// TIA Portal V20 export
TYPE "type_emRelations_em11_sequence"
// stored: Access Published, Namespace Unit1
   STRUCT
      weightCheck : Struct
         jobs : "LAF_typeJobs";
         sequence : "LAF_typeSequence";
         selectJobStatus { S7_SetPoint := 'True'} : Array[0..10] of "LAF_typeJobStatus";
         "step" : "LER_typeStep";
         jobInterface : Struct
            loadJob2 : "LER_typeJobInterface";
            inspectionJob3 : "LER_typeJobInterface";
            unloadJob4 : "LER_typeJobInterface";
         END_STRUCT;
         homeCheck : Struct
            partNoDetect { ExternalWritable := 'False'} : Bool;
            partDetect { ExternalWritable := 'False'} : Bool;
         END_STRUCT;
      END_STRUCT;
   END_STRUCT;
   // // weightCheck."step".action1[101] : Step[101] : JOB[1] Condition
   // // weightCheck."step".action1[110] : Step[110] : Stage Lift Down
   // // weightCheck."step".action1[190] : Step[190] : JOB[1] Step End
   // // weightCheck."step".action1[201] : Step[201] : JOB[2] Condition
   // // weightCheck."step".action1[210] : Step[210] : Weight Check Loading Request => Transfer PP Right
   // // weightCheck."step".action1[230] : Step[230] : Stage Lift Up
   // // weightCheck."step".action1[240] : Step[240] : Weight Check Loading Check => Transfer PP Right
   // // weightCheck."step".action1[250] : Step[250] : Weight Check JR Detection Check
   // // weightCheck."step".action1[290] : Step[290] : JOB[2] Step End
   // // weightCheck."step".action1[301] : Step[301] : JOB[3] Condition
   // // weightCheck."step".action1[310] : Step[310] : Stage Lift Down
   // // weightCheck."step".action1[330] : Step[330] : Weight Check
   // // weightCheck."step".action1[390] : Step[390] : JOB[3] Step End
   // // weightCheck."step".action1[401] : Step[401] : JOB[4] Condition
   // // weightCheck."step".action1[410] : Step[410] : Stage Lift Up
   // // weightCheck."step".action1[430] : Step[430] : Weight Check Unloading Request => JR Unload P&P
   // // weightCheck."step".action1[431] : Step[431] : Weight Check Unloading Check => JR Unload P&P
   // // weightCheck."step".action1[480] : Step[480] : Stage Lift Down
   // // weightCheck."step".action1[490] : Step[490] : JOB[4] Step End
   // // weightCheck."step".transition1[101] : Step[101] : JOB[1] Condition
   // // weightCheck."step".transition1[110] : Step[110] : Stage Lift Down
   // // weightCheck."step".transition1[190] : Step[190] : JOB[1] Step End
   // // weightCheck."step".transition1[201] : Step[201] : JOB[2] Condition
   // // weightCheck."step".transition1[210] : Step[210] : Weight Check Loading Request => Transfer PP Right
   // // weightCheck."step".transition1[230] : Step[230] : Stage Lift Up
   // // weightCheck."step".transition1[240] : Step[240] : Weight Check Loading Check => Transfer PP Right
   // // weightCheck."step".transition1[250] : Step[250] : Weight Check JR Detection Check
   // // weightCheck."step".transition1[290] : Step[290] : JOB[2] Step End
   // // weightCheck."step".transition1[301] : Step[301] : JOB[3] Condition
   // // weightCheck."step".transition1[310] : Step[310] : Stage Lift Down
   // // weightCheck."step".transition1[330] : Step[330] : Weight Check
   // // weightCheck."step".transition1[390] : Step[390] : JOB[3] Step End
   // // weightCheck."step".transition1[401] : Step[401] : JOB[4] Condition
   // // weightCheck."step".transition1[410] : Step[410] : Stage Lift Up
   // // weightCheck."step".transition1[430] : Step[430] : Weight Check Unloading Request => JR Unload P&P
   // // weightCheck."step".transition1[431] : Step[431] : Weight Check Unloading Check => JR Unload P&P
   // // weightCheck."step".transition1[480] : Step[480] : Stage Lift Down
   // // weightCheck."step".transition1[490] : Step[490] : JOB[4] Step End
END_TYPE
